// TwinCAT 3 PLC project Crane_Control
// ProgramVersion: 3.1.4026.20
// CompilerDefines: VISU_USEPROPERTYINFO
// libraries:
//   Tc2_Standard, * (Beckhoff Automation GmbH)
//   Tc2_System, * (Beckhoff Automation GmbH)
// project tree:
//   Bachelor 2026/Enumeration/ E_PressureFeedback.TcDUT (not stored)
//   Bachelor 2026/FB/ FB_ControllerMode.TcPOU (not stored), FB_Filter.TcPOU, FB_InitialPosition.TcPOU (not stored), FB_JoystickScaler.TcPOU (not stored), FB_Normalization.TcPOU (not stored), FB_CylinderScaling.TcPOU (not stored), FB_PF_GradientFiltered.TcPOU (not stored), FB_ValveControl.TcPOU
//   Bachelor 2026/FB/Pressure Feedback to be deleted/ FB_PF_AreaRatio.TcPOU (not stored), FB_PressureFeedback_Simple.TcPOU (not stored)
//   Bachelor 2026/HMI/ HMI.TcVIS
//   Bachelor 2026/PRG/Autoramp/ PRG_AutoRamp_AreaRatio.TcPOU (not stored), PRG_AutoRamp_GradientFiltered.TcPOU (not stored)
//   Bachelor 2026/PRG/Manual Driving to be deleted/ PRG_ManualDriving.TcPOU (not stored), PRG_ManualDriving_AreaRatioPF.TcPOU, PRG_ManualDriving_PF_Home.TcPOU
//   Bachelor 2026/PRG/ PRG_ControllerMode.TcPOU (not stored), PRG_Manual_PF_Gradient.TcPOU (not stored), PRG_Output.TcPOU, PRG_Filter.TcPOU, PRG_ScaledInputs.TcPOU (not stored)
//   Bachelor 2026/PRG/Testing/ fU_Testing.TcPOU (not stored), RampfUTest.TcPOU (not stored)
//   / GlobalTextList.TcGTLO (not stored), MAIN.TcPOU (not stored), PlcTask.TcTTO (not stored), Visualization Manager.TcVMO (not stored)
//   GVL/ G_Enables.TcGVL, G_FilterConstants.TcGVL (not stored), G_Filtered.TcGVL (not stored), G_Init.TcGVL (not stored), G_Inputs.TcGVL, G_Mode.TcGVL, G_OPC.TcGVL (not stored), G_Output.TcGVL (not stored), G_Parameter.TcGVL (not stored)
//   OLD/OLD Enumeration/ E_Mode.TcDUT (not stored), E_Motion.TcDUT (not stored)
//   OLD/OLD Function Blocks/ FB_AutoClock.TcPOU, FB_ControlSignal.TcPOU (not stored), FB_Derivator.TcPOU (not stored), FB_FeedForward.TcPOU (not stored), FB_FeedForward_NonLinear.TcPOU (not stored), FB_Filtering.TcPOU (not stored), FB_Home.TcPOU (not stored), FB_InitialPos.TcPOU (not stored), FB_Integrator.TcPOU (not stored), FB_JoystickInputScaling.TcPOU (not stored), FB_KvFF.TcPOU (not stored), FB_MotionRef.TcPOU (not stored), FB_NaiveFF.TcPOU (not stored), FB_Normalize.TcPOU (not stored), FB_PID.TcPOU (not stored), FB_PositionInputScaling.TcPOU (not stored), FB_PressureFeedback.TcPOU (not stored), FB_RunClock.TcPOU, FB_Running.TcPOU (not stored), FB_ValveOutput.TcPOU (not stored)
//   OLD/OLD Programs/ P_ControlBlock.TcPOU (not stored), P_FeedForward.TcPOU (not stored), P_Filtering.TcPOU (not stored), P_Inputs.TcPOU, P_Modes.TcPOU (not stored), P_Output.TcPOU (not stored), P_PID.TcPOU (not stored), P_RunClock.TcPOU (not stored)
// real-time tasks:
//   TASK PlcTask: cycle T#1ms, priority 20, ADS port 350
// I/O:
//   DEVICE Device 1 (EtherCAT), AmsNetId 192.168.0.204.4.1
//     RIO (EK1100) [EK1100 EtherCAT Coupler (2A E-Bus)]
//       DI (EL1008) [EL1008 8Ch. Dig. Input 24V, 3ms]
//       DO (EL2008) [EL2008 8Ch. Dig. Output 24V, 0.5A]
//       AI1 (EL3068) [EL3068 8Ch. Ana. Input 0-10V]
//       AI2 (EL3068) [EL3068 8Ch. Ana. Input 0-10V]
//       AI3 (EL3174) [EL3174 4Ch. Ana. Input +/-10V Diff., +/-20mA SingleEnded, 16 Bit]
//       AO (EL4104) [EL4104 4Ch. Ana. Output 0-10V, 16bit]
//       End Cap (EL9011) [EL9011 End Terminal]
// variable links:
//   Crane_Control/Crane_Control Instance <-> Device 1 (EtherCAT)/RIO (EK1100)/AI1 (EL3068)
//     PlcTask Inputs/G_Inputs.nRawJoystick <-> AI Standard Channel 2/Value
//     PlcTask Inputs/G_Inputs.nRawPistonPosition <-> AI Standard Channel 3/Value
//     PlcTask Inputs/G_Inputs.nRawSpoolPosition <-> AI Standard Channel 4/Value
//   Crane_Control/Crane_Control Instance <-> Device 1 (EtherCAT)/RIO (EK1100)/AI2 (EL3068)
//     PlcTask Inputs/G_Inputs.nRawPa <-> AI Standard Channel 4/Value
//     PlcTask Inputs/G_Inputs.nRawPaLower <-> AI Standard Channel 5/Value
//     PlcTask Inputs/G_Inputs.nRawPb <-> AI Standard Channel 6/Value
//     PlcTask Inputs/G_Inputs.nRawPs <-> AI Standard Channel 1/Value
//   Crane_Control/Crane_Control Instance <-> Device 1 (EtherCAT)/RIO (EK1100)/AO (EL4104)
//     PlcTask Outputs/G_Output.nValveOutput <-> AO Output Channel 1/Analog output
//   Crane_Control/Crane_Control Instance <-> Device 1 (EtherCAT)/RIO (EK1100)/DI (EL1008)
//     PlcTask Inputs/G_Inputs.bAuto <-> Channel 1/Input
//     PlcTask Inputs/G_Inputs.bManual <-> Channel 2/Input
//     PlcTask Inputs/G_Inputs.bStartButton <-> Channel 3/Input
//     PlcTask Inputs/G_Inputs.bStopButton <-> Channel 4/Input
//   Crane_Control/Crane_Control Instance <-> Device 1 (EtherCAT)/RIO (EK1100)/DO (EL2008)
//     PlcTask Outputs/G_Output.bGreenLight <-> Channel 1/Output
//     PlcTask Outputs/G_Output.bRedLight <-> Channel 2/Output
//     PlcTask Outputs/G_Output.bRunning <-> Channel 3/Output

// ---- GVL/G_Enables.TcGVL
{attribute 'qualified_only'}
// BOOL: True/False

VAR_GLOBAL
	
	// Control Enables
	bEnablePID 		: BOOL; 	// Enable PID Control
	bEnableFF 		: BOOL; 	// Enable FeedForward	
	bEnablePFB		: BOOL; 	// Enable Pressure Feedback
	bEnableU 		: BOOL; 	// Enable Signal to Valve

	bCharTesting	: BOOL; 	// Enable Characteristic testing
	bMove2Home		: BOOL; 	// Enable Home-function
	
	// No Function
	bEnableComp 	: BOOL; 	// Driving with Compensator
	
	// Enumerators
	nModeSelect		: E_Motion; // Motion Reference
	
END_VAR

// ---- GVL/G_Inputs.TcGVL
{attribute 'qualified_only'} // Variable needs to be used with GVL-name

// INT: [-32768, 32767]	
// BOOL: True/False
// %I* assigns next available memory adress in Twincat (In)

VAR_GLOBAL
	// Mode Selection
	bManual 			AT %I* : BOOL; 		// Manual mode controller
	bAuto	 			AT %I* : BOOL;		// Auto mode controller
	bStartButton		AT %I* : BOOL; 		// Start button
	bStopButton			AT %I* : BOOL;		// Stop button
	
	// Raw Pressure Values
	nRawPa 				AT %I*	: INT;		// Pressure cap side
	nRawPb				AT %I*	: INT;		// Pressure rod side
	nRawPs				AT %I*	: INT;		// Pressure supply
	nRawPaLower			AT %I* 	: INT;		// Pressure under counterbalance valve
	
	// Raw Position Values
	nRawPistonPosition 	AT %I*	: INT;		// Piston position
	nRawJoystick		AT %I*	: INT;		// Joystick Y-position
	nRawFlowSensor		AT %I*	: INT;		// Flow sensor
	nRawSpoolPosition	AT %I*	: INT;		// Spool position
END_VAR

// ---- GVL/G_Mode.TcGVL
{attribute 'qualified_only'}
// BOOL: True/False

VAR_GLOBAL // Different modes true/false
	bRunning : BOOL;		// System running
	bManual : BOOL;			// Manual mode
	bAuto : BOOL;			// Auto mode
END_VAR

// ---- Bachelor 2026/FB/FB_Filter.TcPOU
FUNCTION_BLOCK FB_Filter
// SINT: Integer [-128, 127]
// LREAL: Long Real decimal number
// USINT: Integer, strictly positive [0,255]

// Input variables
VAR_INPUT
	FilterMode: SINT;			// 0/1 
	Signal: LREAL; 				// Input signal
	Num: LREAL; 				// Filter constant
	Den: LREAL; 				// Filter constant
	Initial: LREAL; 			// Filter constant
END_VAR

// Output variables
VAR_OUTPUT
	Signal_Unfiltered: LREAL;	// Unfiltered signal
	Signal_Filtered: LREAL;		// Filtered signal
END_VAR

// Variables
VAR
	InitialCondition: USINT; 	// Initial condition load (start value)
	FilterState: LREAL; 		// Filter state/memory (how the filter works)
END_VAR


CASE FilterMode OF
    SS_INITIALIZE:								
        InitialCondition := 1;							// If FilterMode = SS_INITIALIZE (0), set InitialCondition = 1 (reset filter)

    SS_STEP:
        IF InitialCondition <> 0 THEN					// If InitialCondition is not equal to zero, set initial filter values
            FilterState := Initial;
            InitialCondition := 0;						// set InitialCondition = 0 after reset
        END_IF;

        Signal_Unfiltered := Signal;					// Unfiltered input signal
        Signal_Filtered   := Num * FilterState;			// Filtered output
        
        FilterState := Signal - (Den * FilterState); 	// Update filter state (negative feedback)
		
		// Filter adds a percentage of old signal value to the new value (according to value of Den). 
		// This makes the filter calculate slowly and wont be able to fit big spikes/noice in unfiltered signal.
END_CASE;

END_FUNCTION_BLOCK

// ---- Bachelor 2026/FB/FB_ValveControl.TcPOU
FUNCTION_BLOCK FB_ValveControl
// LREAL: Long Real decimal number
// INT: [-32768, 32767]	
// BOOL: True/False

// Input variables
VAR_INPUT
	bEnable 			: BOOL; 	// Enable signal
	fNormalizedInput 	: LREAL;	// Normalized input-data
END_VAR

// Output variables
VAR_OUTPUT
	nOutput : INT; 
END_VAR

// Variables
VAR		
	// [3V, 9V]: (Voltage/10)*32767 
	nOffset 	: LREAL := 19630.0; 	// Closed valve	6V		
	nMaxValue	: LREAL := 29460.0; 	// Max value valve 9V		
	nMinValue 	: LREAL :=  9830.0; 	// Min value valve 3V	
	nTempOutput : LREAL; 				// Temporary output
END_VAR


IF fNormalizedInput > 0.0 THEN													// Signal to set spool at wanted position > 0.0
    nTempOutput := nOffset + (fNormalizedInput * (nMaxValue - nOffset));		// Converts wanted output for valve [19630, 29460] (positive direction)
ELSE																			// Signal to set spool at wanted position < 0.0
    nTempOutput := nOffset + (fNormalizedInput * (nOffset - nMinValue));		// Converts wanted output for valve [9830, 19630] (negative direction)
END_IF

nOutput := LREAL_TO_INT(SEL(bEnable, nOffset, nTempOutput));	// If bEnable is false, output = nOffset (closed valve). 
																// If bEnable is true, output = nTempOutput

END_FUNCTION_BLOCK

// ---- Bachelor 2026/PRG/Manual Driving to be deleted/PRG_ManualDriving_AreaRatioPF.TcPOU
PROGRAM PRG_ManualDriving_AreaRatioPF

VAR
    // Styring og Tilstand
    bReturning         : BOOL;                 // True når Home-sekvens kjører
    ePFMode            : E_PressureFeedback := E_PressureFeedback.PF_ON; // PF alltid på som standard
    
    // FB Instanser
    fbInitialPos       : FB_InitialPos;        // Lagrer startposisjon
    fbReturnTimer      : TON;                  // Timer for 5s hold (Home)
    fbAreaRatioDamping : FB_PF_AreaRatio;      // DEN NYE AREA RATIO FB-en
    
    // Innstillinger for Home-funksjon (Myk start/stopp)
    fHomeTimer         : LREAL;                // Sekunder for oppramping
    fHomeRampTime      : LREAL := 4.0;         // Tid til full fart
    fHomeMaxSpeed      : LREAL := 0.15;        // Toppfart Home
    fCycleTime         : LREAL := 0.01;        // 10ms syklus
    
    // Hjelpevariabler
    fSpeed             : LREAL;                // Mellomverdi for fart
    fDistance          : LREAL;                // Avstand til 0.01
END_VAR

// 1. Oppdater initial posisjon (for statistikk/logging)
fbInitialPos(
    bEnable := G_Inputs.bStartButton AND G_Mode.bRunning,
    fCurrentPos := G_OPC.fPistonPosition
);

// 2. Return Home Logikk (Hold knappen i 5s)
fbReturnTimer(IN := G_Inputs.bStartButton AND G_Mode.bRunning, PT := T#5S);
IF fbReturnTimer.Q THEN
    bReturning := TRUE;
END_IF

// Avbryt Home hvis joysticken beveges mer enn 10%
IF ABS(G_OPC.fJoystick) > 0.1 THEN 
    bReturning := FALSE;
END_IF

// 3. Kjøre-logikk (Home vs Manuelt)
IF bReturning THEN
    // Myk oppstart-timer
    fHomeTimer := fHomeTimer + fCycleTime;
    fDistance := ABS(G_OPC.fPistonPosition - 0.01); 
    
    IF G_OPC.fPistonPosition > 0.01 THEN
        // Rampe opp fart
        fSpeed := (fHomeTimer / fHomeRampTime) * fHomeMaxSpeed;
        
        // Bremsing nær målet (Limit sikrer minimumsfart for å overvinne friksjon)
        fSpeed := LIMIT(0.12, fDistance * 2.0, fSpeed); 
        
        G_OPC.fU := LIMIT(0.0, fSpeed, fHomeMaxSpeed);
    ELSE
        // Vi er hjemme
        G_OPC.fU := 0.0;
        bReturning := FALSE;
        fHomeTimer := 0.0;
    END_IF
ELSE
    fHomeTimer := 0.0;
    
    IF G_Mode.bManual AND G_Mode.bRunning THEN
        // Inverterer joystick slik som i ditt originale script
        G_OPC.fU := -G_OPC.fJoystick;
    ELSE
        G_OPC.fU := 0.0; 
    END_IF
END_IF

// 4. Bruk den nye Area Ratio Pressure Feedback blokken
fbAreaRatioDamping(
    fPa         := G_OPC.fPa,
    fPb         := G_OPC.fPb,
    fJoystick   := G_OPC.fU,
    bEnable     := (ePFMode = E_PressureFeedback.PF_ON),
    fDp         := 0.065,         // Diameter stempel fra din FB
    fDr         := 0.035,         // Diameter stang fra din FB
    fKf         := 0.00001,       // Gain
    fTf         := 0.5,           // Filtertid
    fU_Out      => G_OPC.fU       // Skriver filtrert verdi tilbake til fU
);

// 5. Ventil Dødsone Kompensasjon
IF G_OPC.fU > 0.0 THEN
    G_OPC.fU := G_OPC.fU + G_Parameter.fDeadUp;
ELSIF G_OPC.fU < 0.0 THEN
    // Bruker din originale logikk: G_OPC.fU - fDeadDown (Sjekk fortegn i GVL!)
    G_OPC.fU := G_OPC.fU - G_Parameter.fDeadDown;
END_IF

// 6. Endelig sikkerhetsbegrensning
G_OPC.fU := LIMIT(-1.0, G_OPC.fU, 1.0);

END_PROGRAM

// ---- Bachelor 2026/PRG/Manual Driving to be deleted/PRG_ManualDriving_PF_Home.TcPOU
PROGRAM PRG_ManualDriving_PF_Home
VAR
    bReturning        : BOOL;                	// True when returning home
    ePFMode           : E_PressureFeedback;  	// PF mode (ON/OFF)
    
    fSelectedPressure : LREAL;               	// Pa/Pb based on direction (Pb for positive direction)
	fDistance : LREAL;						 	// Distance used for breaking in return-home mode
    
    fbInitialPos      : FB_InitialPos;      	// FB for initial position
    fbReturnTimer     : TON;                 	// Timer
    fbDamping         : FB_PressureFeedback_Simple; 	// Pressure feedback
END_VAR


// Updates initial position when start button is pushed.
fbInitialPos(
    bEnable := G_Inputs.bStartButton AND G_Mode.bRunning,
    fCurrentPos := G_OPC.fPistonPosition
);

// If start button is held for 5s, return home
fbReturnTimer(IN := G_Inputs.bStartButton AND G_Mode.bRunning, PT := T#5S);
IF fbReturnTimer.Q THEN
    bReturning := TRUE;
END_IF
// Cancel return-home if joystick is activated 
IF ABS(G_OPC.fJoystick) > 0.1 THEN 
    bReturning := FALSE;
END_IF



// HOME uten bremsing (IKKE SLETT FØR TESTING AV BREMSING)
// IF bReturning THEN
//     // --- HOME MODE ---
//     IF G_OPC.fPistonPosition > 0.01 THEN
//         G_OPC.fU := 0.4; // Kjørehastighet hjem 0.15 originalt
//     ELSE
//         G_OPC.fU := 0.0;
//         bReturning := FALSE; // Ferdig hjemme
//     END_IF
// ELSE
// 
//     // --- MANUELL MODUS ---
//     IF G_Mode.bManual AND G_Mode.bRunning THEN
//         G_OPC.fU := -G_OPC.fJoystick;
//     ELSE
//         G_OPC.fU := 0.0; // Failsafe
//     END_IF
// END_IF
// 





//////////////////////////////////////////TEST HOME MED BREMSING
IF bReturning THEN
    fDistance := ABS(G_OPC.fPistonPosition - 0.01); // Calculates distance to home

    IF G_OPC.fPistonPosition > 0.01 THEN 
        G_OPC.fU := fDistance * 4.0; // Change number for early/late breaking (0.4: breaking starts at 0.1m from home)
        G_OPC.fU := LIMIT(0.05, G_OPC.fU, 0.4); // Safety limit for speed
    ELSE
        G_OPC.fU := 0.0;
        bReturning := FALSE;
    END_IF
	
// Manuel mode
ELSE
    IF G_Mode.bManual AND G_Mode.bRunning THEN
        G_OPC.fU := -G_OPC.fJoystick;
    ELSE
        G_OPC.fU := 0.0; 
    END_IF
END_IF
/////////////////////////////////////////////// DELETE AFTER TESTING



// Decides pressure according to movement 
IF G_OPC.fU > 0 THEN
    fSelectedPressure := G_OPC.fPb;
ELSIF G_OPC.fU < 0 THEN
    fSelectedPressure := G_OPC.fPa;
ELSE
    fSelectedPressure := 0.0;
END_IF

// FB for PF
fbDamping(
    bEnable   := (ePFMode = E_PressureFeedback.PF_ON), 
    fInputU   := G_OPC.fU,
    fPressure := fSelectedPressure,
    fOutputU  => G_OPC.fU
);

// Compansates for valve deadband L
IF G_OPC.fU > 0.0 THEN
    G_OPC.fU := G_OPC.fU + G_Parameter.fDeadUp;
ELSIF G_OPC.fU < 0.0 THEN
    G_OPC.fU := G_OPC.fU - G_Parameter.fDeadDown;
END_IF

G_OPC.fU := LIMIT(-1.0, G_OPC.fU, 1.0); // Safety limit

END_PROGRAM

// ---- Bachelor 2026/PRG/PRG_Output.TcPOU
PROGRAM PRG_Output

VAR
	fbValveOutput : FB_ValveControl;
END_VAR

G_Enables.bEnableU := G_Mode.bRunning; // Lagt til senere

// Runs FB with given values
fbValveOutput(
	fNormalizedInput := G_OPC.fU,		// Signal to set spool at wanted position
	bEnable := G_Enables.bEnableU,		// Enable signal
	nOutput => G_Output.nValveOutput	// Output signal to valve
);

// If system is running, set green and red light on controller true. False when not running:
G_Output.bGreenLight := G_Mode.bRunning;
G_Output.bRedLight   := G_Mode.bRunning;

END_PROGRAM

// ---- Bachelor 2026/PRG/PRG_Filter.TcPOU
PROGRAM PRG_Filter

// Variables
VAR
	fbFilterPa : FB_Filter;
	fbFilterPb : FB_Filter;
	fbFilterPs : FB_Filter;
	fbFilterPaLower : FB_Filter;
END_VAR

fbFilterPa(
	FilterMode := 1,
	Signal := G_OPC.fPa, // Unfiltered, normalized pressure 
	
	// Filter constants:
	Num := G_FilterConstants.fPressureFilterNum,
	Den := G_FilterConstants.fPressureFilterDen,
	Initial := G_FilterConstants.fPressureFilterInit,
	
	// Filtered pressure:
	Signal_Filtered => G_Filtered.fPressurePistonSideFiltered,
	Signal_Filtered => G_OPC.fPaFiltered
);

fbFilterPb(
	FilterMode := 1,
	Signal := G_OPC.fPb,
	Num := G_FilterConstants.fPressureFilterNum,
	Den := G_FilterConstants.fPressureFilterDen,
	Initial := G_FilterConstants.fPressureFilterInit,
	
	Signal_Filtered => G_Filtered.fPressureRodSideFiltered,
	Signal_Filtered => G_OPC.fPbFiltered
);

fbFilterPs(
	FilterMode := 1,
	Signal := G_OPC.fPs,
	Num := G_FilterConstants.fPressureFilterNum,
	Den := G_FilterConstants.fPressureFilterDen,
	Initial := G_FilterConstants.fPressureFilterInit,
	
	Signal_Filtered => G_Filtered.fPressureSupplyFiltered,
	Signal_Filtered => G_OPC.fPsFiltered
);

fbFilterPaLower(
	FilterMode := 1,
	Signal := G_OPC.fPaLower,
	Num := G_FilterConstants.fPressureFilterNum,
	Den := G_FilterConstants.fPressureFilterDen,
	Initial := G_FilterConstants.fPressureFilterInit,
	
	Signal_Filtered => G_Filtered.fPressurePaLower,	
	Signal_Filtered => G_OPC.fPaLowerFiltered
);

END_PROGRAM

// ---- OLD/OLD Function Blocks/FB_AutoClock.TcPOU
FUNCTION_BLOCK FB_AutoClock
// LREAL: Long Real decimal number
// BOOL: True/False

// Input variables
VAR_INPUT
	fStart : BOOL; 		// Start timer
	fRunning : BOOL; 	// System is running
	fCycle : LREAL; 	// Time step
END_VAR

// Output variables
VAR_OUTPUT
	fTime : LREAL; 		// Output (time)
END_VAR

	
IF NOT(fStart) OR NOT(fRunning) THEN 	// If start signal is missing or the system is not running, set time to zero
	fTime := 0.0; 
ELSIF fStart AND fRunning THEN 			// If both start signal and system is on. PLS ticks synced into real time
	fTime := fTime + fCycle;		
END_IF

END_FUNCTION_BLOCK

// ---- OLD/OLD Function Blocks/FB_RunClock.TcPOU
FUNCTION_BLOCK FB_RunClock
// LREAL: Long Real decimal number	
// BOOL: True/False

// Input variables
VAR_INPUT
	bStart 		: BOOL; 		// Set to true
	bStop 		: BOOL; 		// Stop button on controller
	fCycleTime  : LREAL; 		// Time step [s]
END_VAR

// Output variables
VAR_OUTPUT
	fTime : LREAL; 		// Output (time)
END_VAR

// Variables
VAR
	bOnOff : BOOL; 		// True/False
END_VAR

IF bStop OR (G_Work.eStatus = E_Status.Off) THEN 	// If stop button is pressed or system is off 
	bOnOff := FALSE; 
	fTime := 0.0; 
ELSIF bOnOff OR bStart THEN 	// If system is online/start button pushed, start timer
	bOnOff := TRUE;
	fTime := fTime + fCycleTime;
END_IF

END_FUNCTION_BLOCK

// ---- OLD/OLD Programs/P_Inputs.TcPOU
PROGRAM P_Inputs
// LREAL: Long Real decimal number

VAR
	fbNormPa :  FB_Normalize;
	fbNormPb :  FB_Normalize;
	fbNormPs :  FB_Normalize;
	fbNormPaLower : FB_Normalize;
	
	fbNormPistonPosition : FB_PositionInputScaling;
	fbNormSpoolPosition : FB_JoystickInputScaling;
	fbJoystick : FB_JoystickInputScaling;	
	fbFlow	: FB_JoystickInputScaling;		

	fPa : LREAL;
	fPb : LREAL;
	fPs : LREAL;
	fPaLower : LREAL;
	
	fPistonPosition : LREAL;
END_VAR

// Runs FBs with given values

fbNormPa(
	nRawInput := G_Inputs.nRawPa,	// Raw value pressure A
	fMaxValue := 400.0, 			// [Bar]
	fNormalizedInput => G_OPC.fPa	// Unfiltered pressure A out from FB (normalized)
);

fbNormPb(
	nRawInput := G_Inputs.nRawPb,	// Raw value pressure B
	fMaxValue := 400.0, 			// [Bar]
	fNormalizedInput => G_OPC.fPb	// Unfiltered pressure B out from FB (normalized)
);

fbNormPs(
	nRawInput := G_Inputs.nRawPs,	// Raw value pressure S
	fMaxValue := 400.0, 			// [Bar]
	fNormalizedInput => G_OPC.fPs 	// Unfiltered pressure S out from FB (normalized)
);

fbNormPistonPosition(
	nRawInput := G_Inputs.nRawPistonPosition,
	
	fMaxInputValue := 16090.0,
	fMinInputValue := 125.0,
	fMaxOutputValue := 0.5,
	fMinOutputValue := 0.0,	
	
	fOutput => G_OPC.fPistonPosMeasured,
	fActual => G_OPC.fPistonPosition
);
	
fbJoystick(
	nRawInput := G_Inputs.nRawJoystick, // Joystick raw y-position
	fMaxValue := 1.0,
	bEnable := (G_Mode.bRunning AND G_Mode.bManual), // Running and manual needs to be on
	
	fMaxInputValue := 14745.0,
	fMinInputValue := 1620.0,
	fNeutralInputValue := 8140.0,
	fNeutralDeadband := 100.0,
	
	fOutput => G_OPC.fJoystick // Joystick output
);

fbNormPaLower(
	nRawInput := G_Inputs.nRawPaLower, 	// Raw pressure A lower
	fMaxValue := 400.0, 				// [Bar]
	fNormalizedInput => G_OPC.fPaLower	// Unfiltered pressure A lower out from FB (normalized)
);

fbNormSpoolPosition(
	nRawInput := G_Inputs.nRawSpoolPosition,
	fMaxValue := 1.0,
	bEnable := TRUE,
	
	fNeutralInputValue := 8355.0,
	fMaxInputValue := 12645.0,
	fMinInputValue := 4071,
	fNeutralDeadband := 15.0,
	
	fOutput => G_OPC.fSpoolPosition
);

fbFlow(
	bEnable := TRUE,
	nRawInput := G_Inputs.nRawFlowSensor,
	fMaxValue := 150.0, // [l/min]
	
	fMaxInputValue := 32767.0,
	fMinInputValue := 0,
	fNeutralInputValue := 15270.0,
	fNeutralDeadband := 25.0,
	
	fOutput => G_OPC.fFlow
);

END_PROGRAM

// ---- Bachelor 2026/HMI/HMI.TcVIS
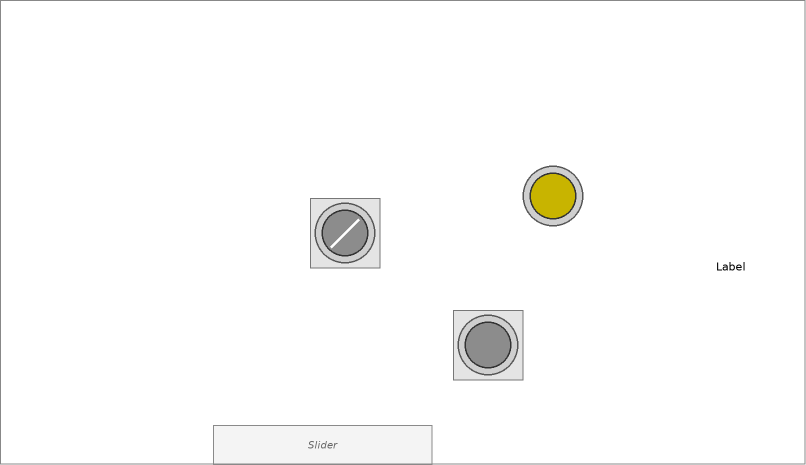
VISUALIZATION HMI  // 806x465
    Lamp1 (518,161 70x70), style: Lamp-Lamp1-Yellow
    RotarySwitch (310,198 70x70), behaviour: TOGGLE, style: Switch-RotarySwitch-Gray
    PushSwitch (453,310 70x70), behaviour: TOGGLE, style: Switch-PushSwitch-Gray
    Label (656,252 150x30), "Label"
    Slider (213,425 219x40), scale 0..100
END_VISUALIZATION
